TYPE ST_MOVE_1 :
STRUCT
	Target:					ST_COORDINATE;
	Override:				LREAL;
	Comment:				STRING(255);
END_STRUCT
END_TYPE

(* stored: Version 1.1.0.1, ProductVersion 3.1.4024.10
   DUT ST_MOVE_1: Id {e23f907f-9111-43e1-b3f3-44913b6916aa} *)
